FUNCTION_BLOCK TAdsReadBySymbolName
VAR
    _Execution : TExecution;
    StateMonitor : TValueMonitor;
    State : INT;

	AmsNetId : T_AmsNetId;
	Port : T_AmsPort;
	SymbolName : STRING;
    ReadDataAddress : PVOID;
    ReadDataLength : UDINT;
    KeepSymbolHandle    : BOOL;  
	SymbolHandle 	   :	DWORD := 0;
    RetryCounter : TCounter;
    
    AdsReadWrite_GetSymHandle : TAdsReadWrite;
    AdsRead_ReadFromSymbol : TAdsRead;
    AdsWrite_ReleaseSymHandle : TAdsWrite;
    
END_VAR
VAR CONSTANT
    sInit          : INT := 0;
    sGetHandle     : INT := 1;
    sReadData      : INT := 2;
    sReleaseHandle : INT := 3;
END_VAR

IF _Execution.Aborting THEN
    State := sInit;
    _Execution.SetAborted();
END_IF

StateMonitor.Test(State);
CASE State OF
    sInit:
        IF _Execution.Starting THEN
            _Execution.SetBusy();
            RetryCounter.Reset();
            IF SymbolHandle = 0 THEN
                State := sGetHandle;
            ELSE
                State := sReadData;
            END_IF
		END_IF
        
    sGetHandle:    
        IF StateMonitor.Changed THEN
            // Get a symbol handle from the runtime...
            AdsReadWrite_GetSymHandle.Execute(
                AmsNetId            := AmsNetId, 
                Port                := Port, 
                IndexGroup          := ADSIGRP_SYM_HNDBYNAME, 
                IndexOffset         := 0, 
                ArgsAddress         := ADR(SymbolName), 
                ArgsLength          := INT_TO_UDINT(LEN(SymbolName)), 
                ReturnValueAddress  := ADR(SymbolHandle), 
                ReturnValueLength   := SIZEOF(SymbolHandle));
        ELSE
            IF AdsReadWrite_GetSymHandle.Execution.Done THEN
                State := sReadData;
			END_IF
            IF AdsReadWrite_GetSymHandle.Execution.Error THEN
                _Execution.SetError(AdsReadWrite_GetSymHandle.Execution.ErrorId);
                SymbolHandle := 0;
                State := sInit;
			END_IF
        END_IF
        
    sReadData: 
        IF StateMonitor.Changed THEN
            // Read the data to from the symbol...
            AdsRead_ReadFromSymbol.Execute(
                AmsNetId        := AmsNetId, 
                Port            := Port, 
                IndexGroup      := ADSIGRP_SYM_VALBYHND, 
                IndexOffset     := SymbolHandle, 
                DataLength      := ReadDataLength, 
                DataAddress     := ReadDataAddress);
        ELSE
            IF AdsRead_ReadFromSymbol.Execution.Done THEN
                IF KeepSymbolHandle THEN
                    _Execution.SetDone();
                    State := sInit;
                ELSE
                    State := sReleaseHandle;
				END_IF

            ELSIF AdsRead_ReadFromSymbol.Execution.Error THEN
                // Detect if it failed due to an online change invalidating the symbol handle...
                IF 
                    AdsRead_ReadFromSymbol.Execution.ErrorId = E_AdsErr.DEVICE_SYMBOLVERSIONINVALID 
                 OR
                    AdsRead_ReadFromSymbol.Execution.ErrorId = E_AdsErr.DEVICE_SYMBOLNOTACTIVE 
                THEN
                    IF RetryCounter.Value > 0 THEN
                        _Execution.SetError(AdsRead_ReadFromSymbol.Execution.ErrorId);
                        SymbolHandle := 0;
                        State := sInit;
                    ELSE
                        RetryCounter.Inc();
                        SymbolHandle := 0;
                        State := sGetHandle;
                    END_IF
                ELSE
                    State := sReleaseHandle;
				END_IF
			END_IF
		END_IF
            
     sReleaseHandle:    
        IF StateMonitor.Changed THEN
            // Release the symbol handle......
            AdsWrite_ReleaseSymHandle.Execute(
                AmsNetId        := AmsNetId, 
                Port            := Port, 
                IndexGroup      := ADSIGRP_SYM_RELEASEHND, 
                IndexOffset     := SymbolHandle, 
                DataLength      := 0, 
                DataAddress     := 0);
        ELSE
            IF AdsWrite_ReleaseSymHandle.Execution.Done THEN
                // Handle write error to the symbol...
                IF AdsRead_ReadFromSymbol.Execution.Error THEN
                    _Execution.SetError(AdsRead_ReadFromSymbol.Execution.ErrorId);
                ELSE
                    _Execution.SetDone();
				END_IF
                SymbolHandle := 0;
                State := sInit;
            ELSIF AdsWrite_ReleaseSymHandle.Execution.Error THEN
                // Handle release handle error...
                _Execution.SetError(AdsWrite_ReleaseSymHandle.Execution.ErrorId);
                SymbolHandle := 0;
                State := sInit;
			END_IF
		END_IF

END_CASE

AdsReadWrite_GetSymHandle();
AdsRead_ReadFromSymbol();
AdsWrite_ReleaseSymHandle();

METHOD Execute : BOOL
VAR_INPUT
	AmsNetId : T_AmsNetId;
	Port : T_AmsPort;
	SymbolName : STRING;
    ReadDataAddress : PVOID;
    ReadDataLength : UDINT;
    KeepSymbolHandle    : BOOL;  
END_VAR
THIS^.AmsNetId          := AmsNetId;
THIS^.Port              := Port;
THIS^.SymbolName        := SymbolName;
THIS^.ReadDataAddress   := ReadDataAddress;
THIS^.ReadDataLength    := ReadDataLength;
THIS^.KeepSymbolHandle  := KeepSymbolHandle;

Execute := _Execution.Start();
END_METHOD

PROPERTY Execution : IExecution
GET
Execution := _Execution;
END_GET
END_PROPERTY

END_FUNCTION_BLOCK

(* stored: Version 1.1.0.1, ProductVersion 3.1.4024.4
   POU TAdsReadBySymbolName: Id {a7401303-b173-4f38-af3b-2ba28c2ac587}, SpecialFunc None
   Method Execute: Id {38e569d7-98bc-4a96-8d29-e1fbbc80730d}
   Property Execution: Id {4e61c5af-ac9c-07a4-34f0-d645f08faa8a}
   Get Get: Id {b8acef8d-80b3-03df-37d9-764d459f3eac} *)
